TYPE T_Lreal : LREAL; END_TYPE

(* stored: Version 1.1.0.1
   DUT T_Lreal: Id {d216545f-a954-4a63-bf95-be8c80f78c6c} *)
